// TIA Portal project "Pick and Place" (V16)
// Vorlageprojekt für das Buch mit Zielsystem S7-1200

(* hardware
DEVICE "S7-1200-Station_1"  S7-1200 Station
   slot 0: "Baugruppenträger_0"  Rack  V1.0
   slot 1: "PLC_1"  CPU 1211C DC/DC/DC  6ES7 211-1AE40-0XB0  V4.1
*)

// ===== PLC "PLC_1"  CPU 1211C DC/DC/DC =====

VAR_GLOBAL   // PLC tag table "Standard-Variablentabelle"
   "m1" AT %M0.0 : Bool;
   "m2" AT %M0.1 : Bool;
   "m3" AT %M0.2 : Bool;
   "Tag_1" AT %I10.0 : Bool;
   "Tag_2" AT %I10.1 : Bool;
   "Tag_3" AT %I10.2 : Bool;
   "Tag_4" AT %I10.3 : Bool;
   "Tag_5" AT %Q10.2 : Bool;
   "Tag_6" AT %I10.6 : Bool;
   "Tag_7" AT %Q10.4 : Bool;
   "Tag_8" AT %Q10.0 : Bool;
   "Tag_9" AT %Q10.1 : Bool;
   "Tag_10" AT %Q10.5 : Bool;
   "Tag_11" AT %I10.5 : Bool;
   "Tag_12" AT %I10.7 : Bool;
   "Tag_13" AT %I10.4 : Bool;
   "Tag_14" AT %Q10.3 : Bool;
END_VAR

VAR_GLOBAL   // PLC tag table "Tag table_1"
   "Start Button 1" AT %I0.0 : Bool;
   "Stop Button 1" AT %I0.1 : Bool;
   "Diffuse Sensor 1" AT %I0.2 : Bool;
   "Diffuse Sensor 2" AT %I0.3 : Bool;
   "Diffuse Sensor 3" AT %I0.4 : Bool;
   "Diffuse Sensor 4" AT %I0.5 : Bool;
   "Diffuse Sensor 5" AT %I0.6 : Bool;
   "Two-Axis Pick & Place 1 (Detected)" AT %I0.7 : Bool;
   "Two-Axis Pick & Place 1 (Moving X)" AT %I1.0 : Bool;
   "Two-Axis Pick & Place 1 (Moving Z)" AT %I1.1 : Bool;
   "Curved Belt Conveyor 1 CW" AT %Q0.0 : Bool;
   "Belt Conveyor (4m) 1" AT %Q0.1 : Bool;
   "Belt Conveyor (6m) 1" AT %Q0.2 : Bool;
   "Two-Axis Pick & Place 1 X" AT %Q0.3 : Bool;
   "Two-Axis Pick & Place 1 Z" AT %Q0.4 : Bool;
   "Two-Axis Pick & Place 1 (Grab)" AT %Q0.5 : Bool;
END_VAR

FUNCTION "MHJ-PLC-Lab-Function-S71200" : Void   // FC9000, SCL
{ S7_Optimized_Access := 'TRUE' }
VERSION : 0.1
   VAR_TEMP
      rdTimeReturn : Int;
      outputTime : DTL;
      SyncVal : Byte;
      forVal : Int;
      forVal_2 : Int;
      Value : Byte;
   END_VAR
   VAR CONSTANT
      CompVal : Byte := 16#34;
      Value_01 : Byte := 16#11;
      Value_01_DW : DWord := 16#A165_D992;
      Value_02_DW : DWord := 16#58BE_4401;
   END_VAR
BEGIN

   #Value:=PEEK(area := 16#82,
        dbNumber := 0,
        byteOffset := 511);
   #Value := #Value + 1;

   POKE(area := 16#82,
        dbNumber := 0,
        byteOffset := 511,
        value := #Value);

   POKE(area:=16#81,
        dbNumber:=0,
        byteOffset:=1016,
        value:=#Value_01_DW);
   POKE(area := 16#81,
        dbNumber := 0,
        byteOffset := 1020,
        value := #Value_02_DW);

   POKE(area := 16#81,
        dbNumber := 0,
        byteOffset := 511,
        value := B#16#00);

   FOR #forVal := 0 TO 120 DO
       FOR #forVal_2:=0 TO 10 DO
           #rdTimeReturn:=RD_SYS_T(#outputTime);
           #rdTimeReturn := WR_SYS_T(#outputTime);
           #rdTimeReturn := RD_SYS_T(#outputTime);
           #rdTimeReturn := WR_SYS_T(#outputTime);
       END_FOR;
       #SyncVal:= PEEK(area := 16#81,
                      dbNumber := 0,
                      byteOffset := 511);
       IF #SyncVal = #CompVal THEN
          GOTO M_1;
       END_IF;
   END_FOR;
   RETURN;

   M_1:
   POKE(area := 16#81,
        dbNumber := 0,
        byteOffset := 511,
        value := B#16#0);
END_FUNCTION

ORGANIZATION_BLOCK "Main"   // OB1, LAD, ProgramCycle
TITLE = "Main Program Sweep (Cycle)"
{ S7_Optimized_Access := 'TRUE' }
VERSION : 0.1
   VAR_INPUT
      Initial_Call : Bool;   // Initial call of this OB
      Remanence : Bool;   // =True, if remanent data are available
   END_VAR
BEGIN

REGION Network 1: Konnektierungsbaustein für PLC-Lab
   // Im Netzwerk 1 wird der Konnektierungsbaustein für PLC-Lab aufgerufen.
   // Dieser Aufruf darf nicht entfernt werden!
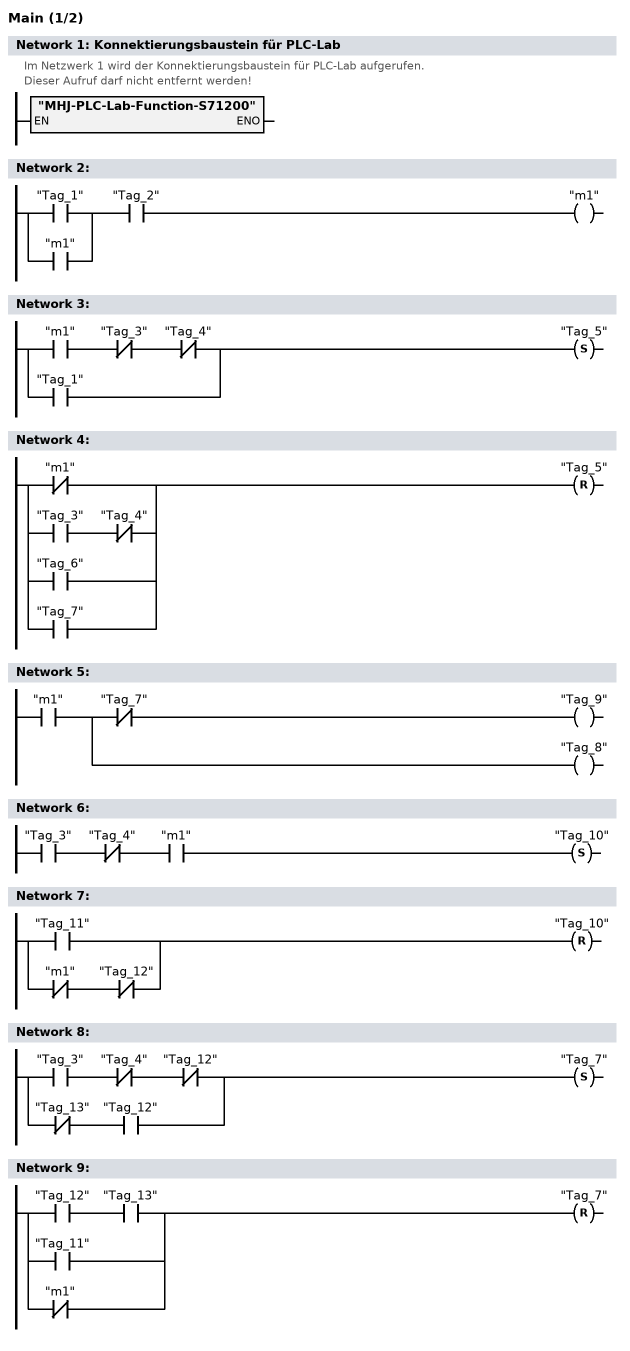
   RUNG wire#powerrail
      "MHJ-PLC-Lab-Function-S71200"()
   END_RUNG
   // the same network as SCL:
   "MHJ-PLC-Lab-Function-S71200"();
END_REGION

REGION Network 2
   RUNG wire#powerrail
      Contact( "Tag_1" )
      wire#w1
      Contact( "Tag_2" )
      Coil( "m1" )
   END_RUNG
   RUNG wire#powerrail
      Contact( "m1" )
   END_RUNG wire#w1
   // the same network as SCL:
   "m1" := ("Tag_1" OR "m1") AND "Tag_2";
END_REGION

REGION Network 3
   RUNG wire#powerrail
      Contact( "m1" )
      I_Contact( "Tag_3" )
      I_Contact( "Tag_4" )
      wire#w1
      S_Coil( "Tag_5" )
   END_RUNG
   RUNG wire#powerrail
      Contact( "Tag_1" )
   END_RUNG wire#w1
   // the same network as SCL:
   IF ("m1" AND NOT "Tag_3" AND NOT "Tag_4") OR "Tag_1" THEN "Tag_5" := TRUE; END_IF;
END_REGION

REGION Network 4
   RUNG wire#powerrail
      I_Contact( "m1" )
      wire#w1
      R_Coil( "Tag_5" )
   END_RUNG
   RUNG wire#powerrail
      Contact( "Tag_3" )
      I_Contact( "Tag_4" )
   END_RUNG wire#w1
   RUNG wire#powerrail
      Contact( "Tag_6" )
   END_RUNG wire#w1
   RUNG wire#powerrail
      Contact( "Tag_7" )
   END_RUNG wire#w1
   // the same network as SCL:
   IF NOT "m1" OR ("Tag_3" AND NOT "Tag_4") OR "Tag_6" OR "Tag_7" THEN "Tag_5" := FALSE; END_IF;
END_REGION

REGION Network 5
   RUNG wire#powerrail
      Contact( "m1" )
      wire#w1
      I_Contact( "Tag_7" )
      Coil( "Tag_9" )
   END_RUNG
   RUNG wire#w1
      Coil( "Tag_8" )
   END_RUNG
   // the same network as SCL:
   "Tag_9" := "m1" AND NOT "Tag_7";
   "Tag_8" := "m1";
END_REGION

REGION Network 6
   RUNG wire#powerrail
      Contact( "Tag_3" )
      I_Contact( "Tag_4" )
      Contact( "m1" )
      S_Coil( "Tag_10" )
   END_RUNG
   // the same network as SCL:
   IF "Tag_3" AND NOT "Tag_4" AND "m1" THEN "Tag_10" := TRUE; END_IF;
END_REGION

REGION Network 7
   RUNG wire#powerrail
      Contact( "Tag_11" )
      wire#w1
      R_Coil( "Tag_10" )
   END_RUNG
   RUNG wire#powerrail
      I_Contact( "m1" )
      I_Contact( "Tag_12" )
   END_RUNG wire#w1
   // the same network as SCL:
   IF "Tag_11" OR (NOT "m1" AND NOT "Tag_12") THEN "Tag_10" := FALSE; END_IF;
END_REGION

REGION Network 8
   RUNG wire#powerrail
      Contact( "Tag_3" )
      I_Contact( "Tag_4" )
      I_Contact( "Tag_12" )
      wire#w1
      S_Coil( "Tag_7" )
   END_RUNG
   RUNG wire#powerrail
      I_Contact( "Tag_13" )
      Contact( "Tag_12" )
   END_RUNG wire#w1
   // the same network as SCL:
   IF ("Tag_3" AND NOT "Tag_4" AND NOT "Tag_12") OR (NOT "Tag_13" AND "Tag_12") THEN "Tag_7" := TRUE; END_IF;
END_REGION

REGION Network 9
   RUNG wire#powerrail
      Contact( "Tag_12" )
      Contact( "Tag_13" )
      wire#w1
      R_Coil( "Tag_7" )
   END_RUNG
   RUNG wire#powerrail
      Contact( "Tag_11" )
   END_RUNG wire#w1
   RUNG wire#powerrail
      I_Contact( "m1" )
   END_RUNG wire#w1
   // the same network as SCL:
   IF ("Tag_12" AND "Tag_13") OR "Tag_11" OR NOT "m1" THEN "Tag_7" := FALSE; END_IF;
END_REGION

REGION Network 10
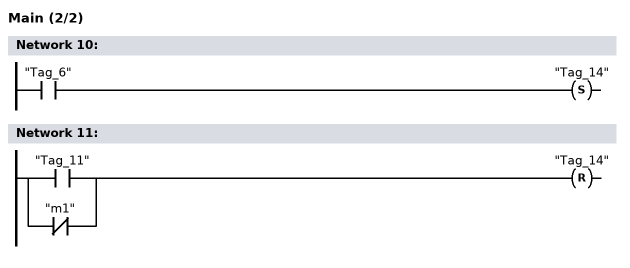
   RUNG wire#powerrail
      Contact( "Tag_6" )
      S_Coil( "Tag_14" )
   END_RUNG
   // the same network as SCL:
   IF "Tag_6" THEN "Tag_14" := TRUE; END_IF;
END_REGION

REGION Network 11
   RUNG wire#powerrail
      Contact( "Tag_11" )
      wire#w1
      R_Coil( "Tag_14" )
   END_RUNG
   RUNG wire#powerrail
      I_Contact( "m1" )
   END_RUNG wire#w1
   // the same network as SCL:
   IF "Tag_11" OR NOT "m1" THEN "Tag_14" := FALSE; END_IF;
END_REGION
END_ORGANIZATION_BLOCK